# EPICS autosave request: ipApp/Db/Metis_M322_settings.req
$(P)$(R):buffMode.VAL
$(P)$(R):readBuff.SCAN
$(P)$(R):unit.VAL
$(P)$(R):focus.VAL
